// TIA Portal V18 export
// export: Created 2026-06-08T17:01:58.7993739Z, ExportSetting WithDefaults, DisplayName Totally Integrated Automation Portal, DisplayVersion V18, DisplayName TIA Portal Openness, DisplayVersion V18, DisplayName TIA Portal Version Control Interface, DisplayVersion V18, DisplayName STEP 7 Professional, DisplayVersion V18, DisplayName STEP 7 Safety, DisplayVersion V18, DisplayName WinCC Professional, DisplayVersion V18
DATA_BLOCK "HMI_DB"   // DB20
{ S7_Optimized_Access := 'FALSE' }
VERSION : 0.1
// stored: AutoNumber true, DBAccessibleFromOPCUA true, IsOnlyStoredInLoadMemory false, IsWriteProtectedInAS false
   VAR
      MAIN_MOVE_F : Bool;
      MAIN_MOVE_R : Bool;
      MAIN_STOP : Bool;
      EMERGENCY : Bool;
      RESET : Bool;
      M1_MOVE_F : Bool;
      M1_MOVE_R : Bool;
      M1_STOP : Bool;
      RESET_COUNTER_1 : Bool;
      M2_MOVE_F : Bool;
      M2_MOVE_R : Bool;
      M2_STOP : Bool;
      RESET_COUNTER_2 : Bool;
      MAIN_FORWARD : Bool;
      MAIN_REVERSE : Bool;
      M1_FORWARD : Bool;
      M1_REVERSE : Bool;
      M2_FORWARD : Bool;
      M2_REVERSE : Bool;
   END_VAR
BEGIN
END_DATA_BLOCK
